PROGRAM MAIN
VAR
	safety				: Safety<CST.MAX_ESTOP>;
	heating				: Heating<CST.MAX_ROOM>;
	standardRoom		: ARRAY[1..5] OF TempTimeRoom;
	receptionRoom		: PassiveRoom;
	conferentionRoom01	: PassiveTempTimeRoom;
	conferentionRoom02	: PassiveTempTimeRoomWithMultipleValves<3>;
	storeRoom01			: TempRoom;
	storeRoom02			: TempRoomWithMultipleSensors<3>;

	dbgInfo				: DebugInfo;
	rtTick				: R_TRIG;
END_VAR

rtTick(CLK :=  Tick(sim.param.nTick), Q => sim.bTick);
Runtime();

METHOD PRIVATE _IO
END_METHOD

END_PROGRAM

(* stored: Version 1.1.0.1
   POU MAIN: Id {46c268e9-fb81-4ca2-9b53-e3c90b600c5e}, SpecialFunc None
   Method _IO: Id {03b676de-555c-400e-bba5-4ba9784520ec} *)
